TYPE PositionAxis_Status :
STRUCT
	STATUS_WORD:UINT;
	POSITION_VALUE:DINT;
END_STRUCT
END_TYPE

(* stored: Version 1.1.0.1, ProductVersion 3.1.4024.12
   DUT PositionAxis_Status: Id {778a3900-b3be-4dc8-873c-b38d849de91f} *)
